FUNCTION Convert_BOOL_TO_INT : BOOL
VAR_INPUT
	in : BOOL;
	out : REFERENCE TO INT;
END_VAR

out := BOOL_TO_INT(in);
Convert_BOOL_TO_INT := TRUE;

END_FUNCTION

(* stored: Version 1.1.0.1, ProductVersion 3.1.4024.12
   POU Convert_BOOL_TO_INT: Id {19ca75a1-9c4a-47b3-9dc9-3a1174b17803}, SpecialFunc None *)
